(* CoDeSys 2.3 export: FTURNOFFK15PUMP.EXP *)

(* POU K15/fTurnOffK15Pump, ST *)
FUNCTION fTurnOffK15Pump :BOOL
VAR_INPUT
	PumpID : USINT;
END_VAR
VAR
END_VAR
	fSetK16Pump(FALSE, PumpID);
END_FUNCTION
